Yaskawa INFORM job: FRONT_WELD_-90ST-1_5040.JBI

/JOB
//NAME FRONT_WELD_-90ST-1_5040
///FOLDERNAME 02-SKRZYNIE_JOBS
//POS
///NPOS 20,20,0,4,0,0
///TOOL 0
///POSTYPE PULSE
///PULSE
C00000=0,-52278,40443,0,6873,1
C00001=0,-52278,40443,-5610,-49281,70968
C00002=0,-42686,23640,-7425,-34877,79161
C00003=14116,-58141,-26117,21696,-5351,66126
C00004=78387,-34691,-23344,93705,-44285,35747
C00005=74588,-16459,-14592,116746,-41260,23896
C00006=70798,-11760,-4995,114918,-37501,24909
C00007=59953,-19295,-11171,117604,-30396,22922
C00008=50123,-24982,-15552,121597,-24133,20342
C00009=32865,-30782,-19575,139278,-14549,10662
C00010=35290,-36639,-28855,139061,-17114,10894
C00011=3902,-39042,-32149,3317,17100,71988
C00012=3902,-39042,-32149,3317,17100,71988
C00013=3166,-35496,-25367,6550,14296,70463
C00014=-17642,-34402,-24928,42875,21231,51544
C00015=-28711,-32549,-24031,51159,27371,46703
C00016=-46392,-26745,-20219,57515,38284,42310
C00017=-48063,-35826,-27915,64657,37344,38904
C00018=-24039,-44019,6278,32369,22109,19464
C00019=0,-52278,40443,0,6873,-1
BC00000=819729
BC00001=872329
BC00002=903040
BC00003=951614
BC00004=975210
BC00005=981280
BC00006=981280
BC00007=981280
BC00008=981280
BC00009=981280
BC00010=981280
BC00011=980954
BC00012=980954
BC00013=980954
BC00014=980956
BC00015=980958
BC00016=980960
BC00017=980954
BC00018=877951
BC00019=774759
///POSTYPE BASE
///RECTAN
///RCONF 0,0,0,0,0,0,0,0,0,0,0,0,0,0,0,0,0,0,0,0,0,0,0,0
P00501=-2.026,0.009,3.534,0.0000,0.0000,0.0000
///RCONF 1,0,0,0,0,0,0,0,0,0,0,0,0,0,0,0,0,0,0,0,0,0,0,0
P00502=-2.023,0.001,1.732,0.0000,0.0000,0.0000
P00503=0.138,-0.044,1.539,0.0000,0.0000,0.0000
P00504=-0.309,-0.010,1.636,0.0000,0.0000,0.0000
//INST
///DATE 2024/05/16 20:52
///ATTR SC,RW
///GROUP1 RB1,BS1
NOP
MOVJ C00000 BC00000 VJ=50.00
MOVJ C00001 BC00001 VJ=50.00
MOVJ C00002 BC00002 VJ=50.00
MOVJ C00003 BC00003 VJ=50.00
MOVJ C00004 BC00004 VJ=50.00
'::::::::::::::::::::::::::::::::
'W56
'::::::::::::::::::::::::::::::::
MOVL C00005 BC00005 V=500.0
SFTON P0501
MACRO1 MJ#(0) ARGF9
MOVL C00006 BC00006 V=166.7 PL=0
ARCON
MOVC C00007 BC00007 V=10.8
SFTOF
SFTON P0502
MOVC C00008 BC00008 V=10.8
MOVC C00009 BC00009 V=10.8
ARCOF
MOVL C00010 BC00010 V=166.7
SFTOF
MOVL C00011 BC00011 V=166.7
'::::::::::::::::::::::::::::::::
'W21
'::::::::::::::::::::::::::::::::
MOVL C00012 BC00012 V=166.7
SFTON P0503
MACRO1 MJ#(0) ARGF9
MOVL C00013 BC00013 V=166.7 PL=0
ARCON
MOVL C00014 BC00014 V=10.8
SFTOF
SFTON P0504
MOVL C00015 BC00015 V=10.8
MOVL C00016 BC00016 V=10.8
ARCOF
MOVL C00017 BC00017 V=250.0
SFTOF
MOVJ C00018 BC00018 VJ=30.00
MOVJ C00019 BC00019 VJ=50.00
END
